// TIA Portal V20 export
VAR_GLOBAL   // PLC tag table "LConSMC_Internal"
END_VAR
VAR_GLOBAL CONSTANT   // user constants
   LCON_TYPE_OF_WINDER_UNWIND_FROM_BELOW : Int := 3;   // Winder configuration parameter "TypeOfWinder"
   LCON_DIAM_CALC_MODE_DIVISION : Int := 0;   // Type of diameter calculation mode
   LCON_DIAM_CALC_MODE_ADDITION : Int := 1;   // Type of diameter calculation mode
   LCON_DIAM_CALC_MODE_INTEGRAL : Int := 2;   // Type of diameter calculation mode
   LCON_DIAM_CALC_MODE_EXTERNAL : Int := 3;   // Type of diameter calculation mode
   LCON_DIAM_CALC_MODE_WEB_LENGTH : Int := 4;   // Type of diameter calculation mode
   LCON_DIAM_CALC_MODE_POSITION : Int := 5;   // Type of diameter calculation mode
   LCON_TYPE_OF_DRIVE_PULL : Int := 0;   // Section drive configuration "typeOfDrive"
   LCON_TYPE_OF_DRIVE_HELD : Int := 1;   // Section drive configuration "typeOfDrive"
   LCON_STATEVAL_MAX_BUFFERLENGTH : UInt := 100;   // max value = 10000
   LCON_STATEVAL_MAX_BUFFERLENGTH_SUB : UInt := 10;
   LCON_STATEVAL_MAX_BUFFERLENGTH_MAIN : UInt := 100;
   LCON_TIMEPERIOD_MODE : UInt := 2;
   LCON_SAMPLEBASED_MODE : UInt := 1;
   LCON_STATEVAL_LEAST_CYCLETIME_IN_MICROSEC : UInt := 125;   // cycle time in µs
   LCON_STATEVAL_MAX_SAMPLINGRATE : UInt := 10000;   // multiple of sampling rate - do not change!
   LCON_STATEVAL_MAX_NUMBER_OF_INPUTSIGNALS : Int := 10;
   LCON_MAX_VALUE_BREAK_POINT_TABLE : Int := 19;   // Maximum length of UDT LConSMC_typeBreakpointTable (0..LCON_MAX_VALUE_BREAK_POINT_TABLE)
   LCON_CONTROL_MODE_V_CONSTANT : Int := 4;   // Winder configuration parameter "controlMode"
   LCON_INVALID_AXIS_TYPE : Int := 0;   // Axis type is invalid
   LCON_PI : LReal := 3.141592;   // Constant PI
   LCON_POSITIONING_AXIS_TYPE : Int := 2;   // Positioning axis
   LCON_SPEED_AXIS_TYPE : Int := 1;   // Speed axis
   LCON_TYPE_OF_WINDER_REWIND_FROM_ABOVE : Int := 0;   // Winder configuration parameter "TypeOfWinder"
   LCON_SYNCHRONOUS_AXIS_TYPE : Int := 3;   // Synchronous axis
   LCON_TYPE_OF_WINDER_REWIND_FROM_BELOW : Int := 1;   // Winder configuration parameter "TypeOfWinder"
   LCON_TYPE_OF_WINDER_UNWIND_FROM_ABOVE : Int := 2;   // Winder configuration parameter "TypeOfWinder"
   LCON_CONTROL_MODE_DANCER_SPEED : Int := 0;   // Winder configuration parameter "controlMode" / Tension control mode "Dancer speed adaption"
   LCON_CONTROL_MODE_TENSION_SPEED : Int := 1;   // Winder configuration parameter "controlMode" / Tension control mode "Load cell speed adaption"
   LCON_CONTROL_MODE_INDIRECT_TENSION : Int := 3;   // Winder configuration parameter "controlMode" / Tension control mode "Indirect tension control via torque adaption"
   LCON_CONTROL_MODE_DRAW_CONTROL : Int := 4;   // Sectional drive configuration parameter "controlMode" / Tension control mode "Draw control"
   LCON_CONTROL_MODE_INDIRECT_TENSION_SPEED_ADAPT : Int := 5;   // Tension control mode "Indirect tension control via speed adaption"
   LCON_CONTROL_MODE_TENSION_TORQUE : Int := 2;   // Winder configuration parameter "controlMode" / Tension control mode "Load cell torque adaption"
END_VAR
